{attribute 'qualified_only'}
{attribute 'strict'}
TYPE HomingMode :
(
	Default := MC_DefaultHoming,
	Direct := MC_Direct,
	ForceCalibration := MC_ForceCalibration,
	ResetCalibration := MC_ResetCalibration
) INT;
END_TYPE

(* stored: Version 1.1.0.1, ProductVersion 3.1.4024.12
   DUT HomingMode: Id {e329794a-7967-49f9-8de8-95a11baa4827} *)
